TYPE XyTableComSubscribe :
STRUCT
  Request : XyTableComRequest; // contains booleans that are used to start a specific sequence.
  Equipment : XyTableComSubscribeEquipment;  // structs for equipment objects which are used by the bridges
  Segments : XyTableComSubscribeSegments;
END_STRUCT
END_TYPE

(* stored: Version 1.1.0.1
   DUT XyTableComSubscribe: Id {fd784cf4-cb32-4e9b-aed0-8ee5c395046a} *)
